(* PLC project Sin nombre, Desconocido Sin nombre 1 *)
(* stored: creationDateTime 2023-04-05T21:43:38, modificationDateTime 2023-04-11T22:24:45 *)

PROGRAM Parcial2CanchonHerreraMayorgaRivera
  VAR
    SensorCounter AT %IX0.0 : BOOL;  (* Sensor infrarrojo que detecta la presencia de una mandarina *)
    StartButton AT %IX0.1 : BOOL;  (* Botón de inicio *)
    StopButton AT %IX0.2 : BOOL;  (* Botón de parado de emergencia *)
    RestartButton AT %IX0.3 : BOOL;  (* Botón de reset *)
    TangerineMotor AT %QX0.0 : BOOL;  (* Motor que mueve la cinta transportadora de mandarinas *)
    BoxMotor AT %QX0.1 : BOOL;  (* Motor que mueve la cinta transportadora de cajas *)
    Stop AT %QX0.2 : BOOL;  (* Indicador de sistema en parado de emergencia *)
    Start AT %QX0.3 : BOOL;  (* Indicador de sistema funcionando *)
  END_VAR
  VAR
    Restart : BOOL;  (* Indicador de sistema en reset *)
    Full : BOOL;  (* Indicador de caja llena *)
    TangerineCounter : INT;  (* Variable con la cantidad de mandarinas en la caja *)
    StopTimer : TIME;  (* Variable con el tiempo transcurrido del sistema en pausa despues de llenada la caja *)
    BoxTimer : TIME;  (* Variable con el tiempo transcurrido del movimiento de la banda de cajas *)
    BoxGoal : BOOL;  (* Indicador del logro de la meta de producción *)
    BoxCounter : INT;  (* Variable con la cantidad de cajas llenadas *)
    CTU0 : CTU;  (* Contador de mandarinas *)
    TON0 : TON;  (* Temporizador de pausa despues de llenada la caja *)
    TON1 : TON;  (* Temporizador de banda transportadora de cajas en movimiento *)
    CTU1 : CTU;  (* Contador de cajas llenadas *)
  END_VAR
  VAR  (* added by the conversion: wires and edge detectors of the diagram *)
    R_TRIG1 : R_TRIG;
    R_TRIG2 : R_TRIG;
  END_VAR

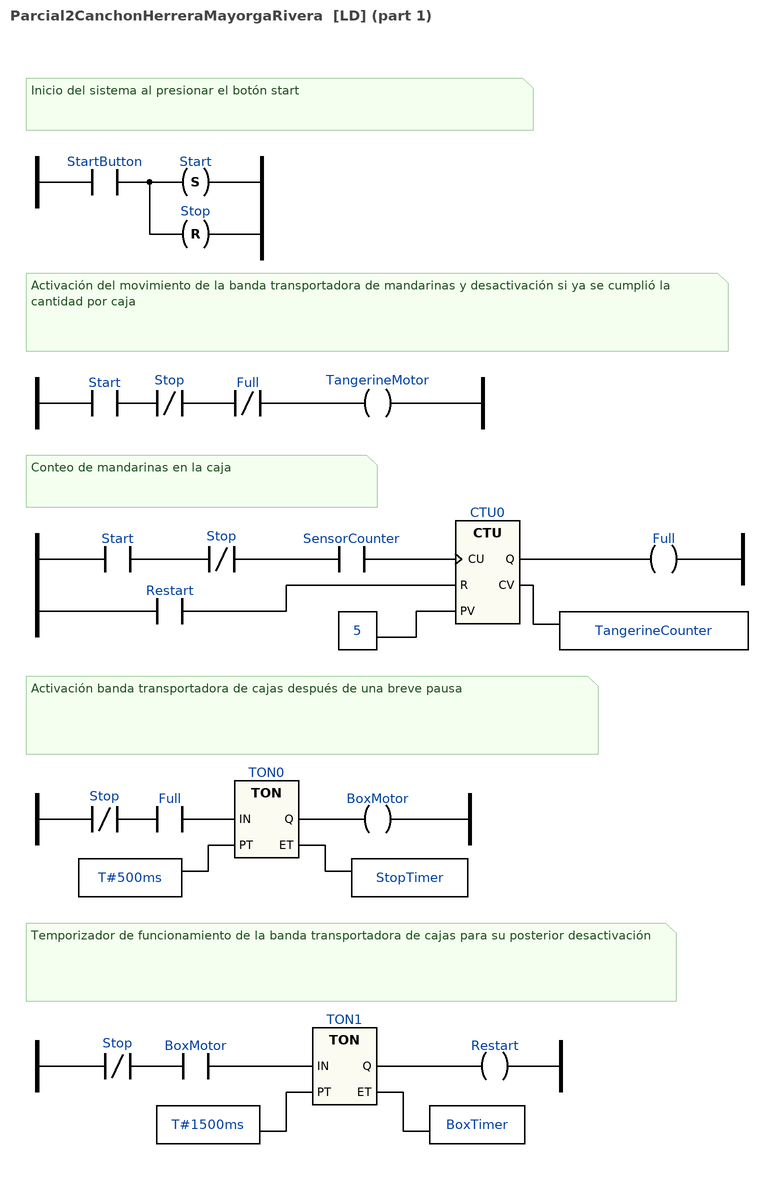
(* LD diagram, written out as Structured Text *)
(* Inicio del sistema al presionar el botón start *)
IF StartButton THEN Start := TRUE; END_IF;
IF StartButton THEN Stop := FALSE; END_IF;
(* Activación del movimiento de la banda transportadora de mandarinas y desactivación si ya se cumplió la cantidad por caja *)
TangerineMotor := Start AND NOT Stop AND NOT Full;
(* Conteo de mandarinas en la caja *)
R_TRIG1(CLK := Start AND NOT Stop AND SensorCounter);
CTU0(CU := R_TRIG1.Q, R := Restart, PV := 5);
Full := CTU0.Q;
TangerineCounter := CTU0.CV;
(* Activación banda transportadora de cajas después de una breve pausa *)
TON0(IN := NOT Stop AND Full, PT := T#500ms);
BoxMotor := TON0.Q;
StopTimer := TON0.ET;
(* Temporizador de funcionamiento de la banda transportadora de cajas para su posterior desactivación *)
TON1(IN := NOT Stop AND BoxMotor, PT := T#1500ms);
Restart := TON1.Q;
BoxTimer := TON1.ET;
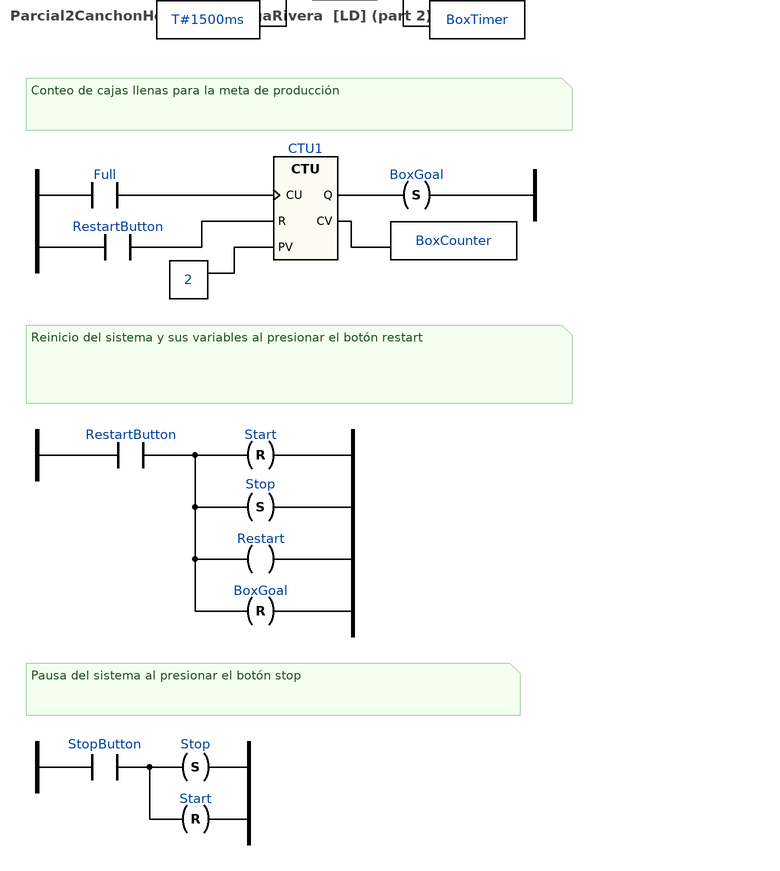
(* Conteo de cajas llenas para la meta de producción *)
R_TRIG2(CLK := Full);
CTU1(CU := R_TRIG2.Q, R := RestartButton, PV := 2);
IF CTU1.Q THEN BoxGoal := TRUE; END_IF;
BoxCounter := CTU1.CV;
(* Reinicio del sistema y sus variables al presionar el botón restart *)
IF RestartButton THEN Start := FALSE; END_IF;
IF RestartButton THEN Stop := TRUE; END_IF;
Restart := RestartButton;
IF RestartButton THEN BoxGoal := FALSE; END_IF;
(* Pausa del sistema al presionar el botón stop *)
IF StopButton THEN Stop := TRUE; END_IF;
IF StopButton THEN Start := FALSE; END_IF;
END_PROGRAM

CONFIGURATION Config0
  RESOURCE Res0 ON PLC
    TASK task0(INTERVAL := T#20ms, PRIORITY := 0);
    PROGRAM instance0 WITH task0 : Parcial2CanchonHerreraMayorgaRivera;
  END_RESOURCE
END_CONFIGURATION
